(* Logix 5000 project; controller Lab1 vendor 1 type 14 code 155 rev 20.12; software revision 20.01 *)

TASK MainTask (continuous, watchdog 500 ms) : MainProgram

MODULES
   Local : vendor 1 type 14 code 155 (PointIO 0, rev 20.12)
      A_In : 1734-IE2V (PointIO 2, rev 3.1, Input RPI 80 ms)
      Stepper_1 : vendor 10 type 150 code 185 (PointIO 5, rev 1.1, Output RPI 50 ms)
      Stepper_2 : vendor 10 type 150 code 185 (PointIO 6, rev 1.1, Output RPI 50 ms)
      Discrete_IO : Embedded (PointIO 1, rev 20.11, Output RPI 20 ms)
      A_Out : 1734-OE2V (PointIO 3, rev 3.1, Output RPI 80 ms)
      HSC : vendor 1 type 109 code 13 (PointIO 4, rev 3.1, Output RPI 80 ms)
END_MODULES

PROGRAM MainProgram   (* main routine MainRoutine *)
VAR
   AnalogVoltage : INT := 1;
   VAR0 : BOOL;
   VAR1 : BOOL;
   VAR2 : BOOL;
   VAR3 : BOOL;
END_VAR

ROUTINE MainRoutine   (* ladder *)
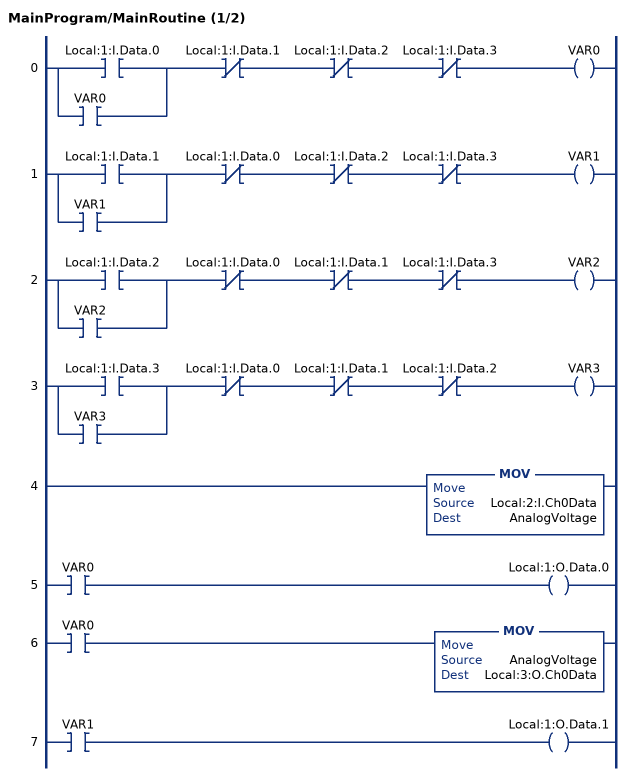
   0: [XIC(Local:1:I.Data.0) ,XIC(VAR0) ]XIO(Local:1:I.Data.1)XIO(Local:1:I.Data.2)XIO(Local:1:I.Data.3)OTE(VAR0);
   1: [XIC(Local:1:I.Data.1) ,XIC(VAR1) ]XIO(Local:1:I.Data.0)XIO(Local:1:I.Data.2)XIO(Local:1:I.Data.3)OTE(VAR1);
   2: [XIC(Local:1:I.Data.2) ,XIC(VAR2) ]XIO(Local:1:I.Data.0)XIO(Local:1:I.Data.1)XIO(Local:1:I.Data.3)OTE(VAR2);
   3: [XIC(Local:1:I.Data.3) ,XIC(VAR3) ]XIO(Local:1:I.Data.0)XIO(Local:1:I.Data.1)XIO(Local:1:I.Data.2)OTE(VAR3);
   4: MOV(Local:2:I.Ch0Data,AnalogVoltage);
   5: XIC(VAR0)OTE(Local:1:O.Data.0);
   6: XIC(VAR0)MOV(AnalogVoltage,Local:3:O.Ch0Data);
   7: XIC(VAR1)OTE(Local:1:O.Data.1);
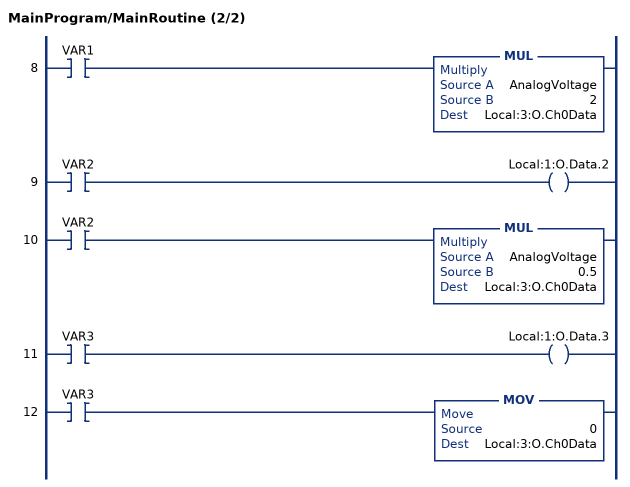
   8: XIC(VAR1)MUL(AnalogVoltage,2,Local:3:O.Ch0Data);
   9: XIC(VAR2)OTE(Local:1:O.Data.2);
   10: XIC(VAR2)MUL(AnalogVoltage,0.5,Local:3:O.Ch0Data);
   11: XIC(VAR3)OTE(Local:1:O.Data.3);
   12: XIC(VAR3)MOV(0,Local:3:O.Ch0Data);
END_ROUTINE
END_PROGRAM
